FUNCTION_BLOCK EcMasterDeviceState IMPLEMENTS IEcTask
VAR_INPUT
END_VAR
VAR_OUTPUT
END_VAR
VAR
	iState : INT;
	masterDeviceState : Tc2_EtherCAT.FB_EcGetMasterDevState;
	_execute: BOOL;
	_done: BOOL;
	_busy: BOOL;
	_error: BOOL;
	_netId: AMSNETID;
END_VAR

CASE iState OF
	0:
		IF _execute THEN
			_done := FALSE;
			_busy := TRUE;
			_error := FALSE;
			masterDeviceState.bExecute := TRUE;
			IF masterDeviceState.bBusy THEN
				iState := 10;
				_execute := false;
			END_IF
		END_IF
	10:
		IF NOT masterDeviceState.bBusy THEN
			IF NOT masterDeviceState.bError THEN
				_done := TRUE;
			ELSE
				_error := TRUE;
			END_IF
			_busy := FALSE;
			masterDeviceState.bExecute := FALSE;
			iState := 0;
		END_IF
END_CASE

masterDeviceState(sNetId := Tc2_System.F_CreateAmsNetId(nIds := NetId));

{warning 'add method implementation '}
METHOD Abort : BOOL
masterDeviceState.bExecute := FALSE;
_busy := FALSE;
_execute := FALSE;
Abort := TRUE;
iState := 0;
END_METHOD

{warning 'add property implementation'}
PROPERTY Busy : BOOL
GET
Busy := _busy;
END_GET
END_PROPERTY

{warning 'add property implementation'}
PROPERTY Done : BOOL
GET
Done := _done;
END_GET
END_PROPERTY

{warning 'add property implementation'}
PROPERTY Error : BOOL
GET
Error := _error;
END_GET
END_PROPERTY

{warning 'add method implementation '}
METHOD Execute : BOOL
IF NOT masterDeviceState.bBusy THEN
	Execute := _execute := true;
END_IF
END_METHOD

PROPERTY MasterDevState : word
GET
MasterDevState := masterDeviceState.nDevState;
END_GET
END_PROPERTY

{warning 'add property implementation'}
PROPERTY NetID : amsnetid
GET
NetID := _netId;
END_GET
SET
_netId := NetID;
END_SET
END_PROPERTY

END_FUNCTION_BLOCK

(* stored: Version 1.1.0.1, ProductVersion 3.1.4024.11
   POU EcMasterDeviceState: Id {03434564-73df-48ce-bbb5-c3f6f90f2964}, SpecialFunc None
   Method Abort: Id {6c42c734-e1e1-4922-82d1-a0798ca263ae}
   Property Busy: Id {a10e39bc-f05e-4616-b97d-ceab9b8dba44}
   Get Get: Id {3f459153-71c3-4d6a-9cf1-9ca7cbc47ac3}
   Property Done: Id {df89d366-63ff-4b11-94d6-c464c84577e4}
   Get Get: Id {bb87c534-8a59-4f05-a54d-543352e1a246}
   Property Error: Id {661079af-deb7-47d7-a0ab-4e504a50e9ee}
   Get Get: Id {895680c8-67d3-4842-8802-42af480e499d}
   Method Execute: Id {4373c8fa-9f21-4d4a-8e60-3d632cd85d99}
   Property MasterDevState: Id {9d52512b-a167-40f0-ac16-ac2dbf3d48cf}
   Get Get: Id {a02a92cb-6fba-48fd-9712-81fc05a9d109}
   Property NetID: Id {3f007876-deb0-4fee-be65-75e6ed2b43b7}
   Get Get: Id {20f563ea-1571-4a38-a3e3-29596a86e3c6}
   Set Set: Id {bd376b00-da43-4d6b-98c7-0b1ed32d2c35} *)
